(* IEC 61131-3 sources: teller/JD_Teller_LC2_V11/Class/Varan_DataMover (part 2) *)

	//check ASY RD DO's
	for i := 0 to VM_DATAMOVER_MAX_DO - 1 do

		//if handle not exists
		if ( a_DO_ASY_RD[ i ].p_Handle = NIL ) then
			exit;
		end_if;

    ud_retries := VaranIn.GetRetryCounter(ud_DOHandle := a_DO_ASY_RD[ i ].p_Handle$UDINT);
    if ( ud_retries <> a_DO_ASY_RD[ i ].us_OldRetryCounter ) then
      VaranIn.RetryCounter += TO_USINT( ud_retries - a_DO_ASY_RD[ i ].us_OldRetryCounter );
      a_DO_ASY_RD[ i ].us_OldRetryCounter := ud_retries$USINT;
		end_if;
	end_for;

	//check ASY WR DO's
	for i := 0 to VM_DATAMOVER_MAX_DO - 1 do

		//if handle not exists
		if ( a_DO_ASY_WR[ i ].p_Handle = NIL ) then
			exit;
		end_if;

    ud_retries := VaranIn.GetRetryCounter(ud_DOHandle := a_DO_ASY_WR[ i ].p_Handle$UDINT);
    if ( ud_retries <> a_DO_ASY_WR[ i ].us_OldRetryCounter ) then
      VaranIn.RetryCounter += TO_USINT( ud_retries - a_DO_ASY_WR[ i ].us_OldRetryCounter );
      a_DO_ASY_WR[ i ].us_OldRetryCounter := ud_retries$USINT;
		end_if;
	end_for;

	//check config DO
	if ( s_ConfigDO.p_Handle <> NIL ) then

		ud_retries := VaranIn.GetRetryCounter(ud_DOHandle := s_ConfigDO.p_Handle$UDINT);
    if ( ud_retries <> s_ConfigDO.us_OldRetryCounter ) then
      VaranIn.RetryCounter += TO_USINT( ud_retries - s_ConfigDO.us_OldRetryCounter );
      s_ConfigDO.us_OldRetryCounter := ud_retries$USINT;
		end_if;
	end_if;

	//check config DO
	if ( s_ConfigWrDO.p_Handle <> NIL ) then

		//if counter changes
    ud_retries := VaranIn.GetRetryCounter(ud_DOHandle := s_ConfigWrDO.p_Handle$UDINT);
    if ( ud_retries <> s_ConfigWrDO.us_OldRetryCounter ) then
      VaranIn.RetryCounter += TO_USINT( ud_retries - s_ConfigWrDO.us_OldRetryCounter );
      s_ConfigWrDO.us_OldRetryCounter := ud_retries$USINT;
		end_if;
	end_if;

//-------------------------------------------------------------------------------------------------
#ifdef VM_DATAMOVER_ISO_TIME
	//check ISO Time DO
	if ( s_ISO_Time_DO.p_Handle <> NIL ) then

    ud_retries := VaranIn.GetRetryCounter(ud_DOHandle := s_ISO_Time_DO.p_Handle$UDINT);
    if ( ud_retries <> s_ISO_Time_DO.us_OldRetryCounter ) then
      VaranIn.RetryCounter += TO_USINT( ud_retries - s_ISO_Time_DO.us_OldRetryCounter );
      s_ISO_Time_DO.us_OldRetryCounter := ud_retries$USINT;
		end_if;
	end_if;
#endif
//-------------------------------------------------------------------------------------------------

	//----------------we have special DO----------------------------------------------------
	if ( us_specialDOCnt <> 0 ) then

		for i := 0 to us_SpecialDOCnt - 1 do

      ud_retries := VaranIn.GetRetryCounter(ud_DOHandle := a_SpecialDO[ i ].p_Handle$UDINT);
      if ( ud_retries <> a_SpecialDO[ i ].us_OldRetryCounter ) then
        VaranIn.RetryCounter += TO_USINT( ud_retries - a_SpecialDO[ i ].us_OldRetryCounter );
        a_SpecialDO[ i ].us_OldRetryCounter := ud_retries$USINT;
			end_if;
		end_for;
	end_if;

END_FUNCTION //GLOBAL Varan_DataMover::GetRetryCounter
//=================================================================================================
//Function to set off all DO's
//=================================================================================================
FUNCTION GLOBAL Varan_DataMover::SetDOsOff
  VAR
    i		: USINT;
  END_VAR

	//check ISO RD DO's
	for i := 0 to VM_DATAMOVER_MAX_DO - 1 do

		//if handle not exists
		if ( a_DO_ISO_RD[ i ].p_Handle = NIL ) then
			exit;
		end_if;

		//set DO off
    VaranIn.DisableDO(ud_DOHandle := a_DO_ISO_RD[ i ].p_Handle$UDINT);
    a_DO_ISO_RD[ i ].b_DOIsRunning := 0;
	end_for;

	//check ISO WR DO's
	for i := 0 to VM_DATAMOVER_MAX_DO - 1 do

		//if handle not exists
		if ( a_DO_ISO_WR[ i ].p_Handle = NIL ) then
			exit;
		end_if;

		//set DO off
    VaranIn.DisableDO(ud_DOHandle := a_DO_ISO_WR[ i ].p_Handle$UDINT);
    a_DO_ISO_WR[ i ].b_DOIsRunning := 0;
	end_for;

	//check ASY RD DO's
	for i := 0 to VM_DATAMOVER_MAX_DO - 1 do

		//if handle not exists
		if ( a_DO_ASY_RD[ i ].p_Handle = NIL ) then
			exit;
		end_if;

		//set DO off
    VaranIn.DisableDO(ud_DOHandle := a_DO_ASY_RD[ i ].p_Handle$UDINT);
    a_DO_ASY_RD[ i ].b_DOIsRunning := 0;
	end_for;

	//check ASY WR DO's
	for i := 0 to VM_DATAMOVER_MAX_DO - 1 do

		//if handle not exists
		if ( a_DO_ASY_WR[ i ].p_Handle = NIL ) then
			exit;
		end_if;

		//set DO off
    VaranIn.DisableDO(ud_DOHandle := a_DO_ASY_WR[ i ].p_Handle$UDINT);
    a_DO_ASY_WR[ i ].b_DOIsRunning := 0;
	end_for;

	//check config DO
	if ( s_ConfigDO.p_Handle <> NIL ) then

		//set DO off
		VaranIn.DisableDO(ud_DOHandle := s_ConfigDO.p_Handle$UDINT);
	end_if;

	//check config WR DO
	if ( s_ConfigWrDO.p_Handle <> NIL ) then

		//set DO off
		VaranIn.DisableDO(ud_DOHandle := s_ConfigWrDO.p_Handle$UDINT);
    s_ConfigWrDO.b_DOIsRunning := 0;
	end_if;

//-------------------------------------------------------------------------------------------------
#ifdef VM_DATAMOVER_ISO_TIME
	//check ISO Time DO
	if ( s_ISO_Time_DO.p_Handle <> NIL ) then

		//set DO off
		VaranIn.DisableDO(ud_DOHandle := s_ISO_Time_DO.p_Handle$UDINT);
	end_if;
#endif
//-------------------------------------------------------------------------------------------------

	//----------------we have special DO----------------------------------------------------
	if ( us_SpecialDOCnt <> 0 ) then

		for i := 0 to us_SpecialDOCnt - 1 do
			//set DO off
			VaranIn.DisableDO(ud_DOHandle := a_SpecialDO[i].p_Handle$UDINT);
      a_SpecialDO[i].b_DOIsRunning := 0;
		end_for;
	end_if;

END_FUNCTION //GLOBAL Varan_DataMover::SetDOsOff
//=================================================================================================
//Function to start ASY List
//=================================================================================================
FUNCTION  Varan_DataMover::StartAsyncList
  VAR
    i			: USINT;
    StartIt : BOOL;
    lbs_ControlReg : t_MoverConfigReg;
  END_VAR

  // switch off dias alive enable
	s_Config.us_ControlReg.DiasAliveEnable	:= FALSE;

	//if we have ASY DO's
	if ( s_Set_ASY_WR.us_DOCount ) then
		for i := 0 to s_Set_ASY_WR.us_DOCount - 1 do
			//start DO single
      if b_PayloadSupport then
        a_DO_ASY_WR[ i ].b_DOIsRunning.StartRequest := TRUE;
      else
      a_DO_ASY_WR[ i ].p_Handle^.ucCtrlStat := VaranIn.SetRunStatus(VARAN_DO_SINGLE_RUN);
      end_if;
		end_for;
	end_if;

  StartIt := FALSE;
	//if we have ASY code
	if ( ui_ASYByteCount ) then
  	//start async list
    s_Config.us_ControlReg.AsyncListEnable	:= TRUE;
    StartIt := TRUE;
  else
  	//don't start async list
    s_Config.us_ControlReg.AsyncListEnable	:= FALSE;

    // if there is no ASY code => don't wait for anything
    us_Wait := 0;
  end_if;
  lbs_ControlReg := s_Config.us_ControlReg;

  if ( lbs_ControlReg.AdminEnable = TRUE ) then
    b_AdminStarted := TRUE;
    us_ControlRd.AdminActive := TRUE;
    StartIt := TRUE;
  end_if;

  if StartIt then
    s_ConfigWrDO.p_DataWrite^ := lbs_ControlReg;

    // reset flag for starting admin task
    IF lbs_ControlReg.AdminEnable = TRUE THEN
      s_Config.us_ControlReg.AdminEnable := FALSE;
    END_IF;

    if b_PayloadSupport then
      s_ConfigWrDO.b_DOIsRunning.StartRequest :=TRUE;
    else
    s_ConfigWrDO.p_Handle^.ucCtrlStat := VaranIn.SetRunStatus(VARAN_DO_SINGLE_RUN);
    end_if;
		us_Wait := 1;		//because otherwise we have old async ready bit

	end_if;

END_FUNCTION // Varan_DataMover::StartAsyncList
//[#ENGLISH]
//=================================================================================================
//Function to add an ISO Rd Enable
//=================================================================================================
//[>ud_add]address of access
//[>ud_length]length of data
//[>p_data]address of pointer variable to save data address
//[>p_enable]address of pointer to start single call
FUNCTION GLOBAL Varan_DataMover::AddRdISOEnable
  VAR_INPUT
    ud_add			: UDINT;
    ud_length		: UDINT;
    p_data			: ^void;
    p_enable		: ^USINT;
      ud_Priority 	: HDINT;
    p_DataAddr : ^HDINT;
		p_UserDOHandle 	: ^UDINT;
  END_VAR
  VAR_OUTPUT
    sd_retval		: DINT;
  END_VAR
  VAR
    p_Mov			: ^t_StructMoveEn;
    ud_dest_add		: UDINT;
    ud_en_add		: UDINT;
  END_VAR

	//get memory for single call
  sd_retval := GetMemoryISORd(p_add         := #ud_dest_add
                              , p_data	:= p_data
                              , ud_len	:= ud_length
                              , ud_Priority := ud_Priority
                            , p_UserDOHandle:= p_UserDOHandle
                              );

	if ( sd_retval <> VARANMANAGER_OK ) then
		return;
	end_if;

  //give back the address if requested
  if p_DataAddr then
    p_DataAddr^ := ud_dest_add;
  end_if;

	//for enable byte
	sd_retval := GetMemoryISOWr	( p_add		:= #ud_en_add
                              , p_data	:= p_enable
                              , ud_len	:= 1
                              );

	if ( sd_retval <> VARANMANAGER_OK ) then
		return;
	end_if;

	//give back address of enable byte
	( ( ( p_enable$^UDINT )^ )$^USINT )^ := 0;

	//save opcodes in class
	if ( p_ISOMoverCode = NIL ) then
		//allocate memory
		p_ISOMoverCode$^void := To_StdLib.Malloc( s_Set_ISO_RD.ui_DPRAMSize + s_Set_ISO_WR.ui_DPRAMSize );

		if ( p_ISOMoverCode  = NIL ) then
			State := _MemoryFault;
			sd_retval := -103;
			VaranIn.SetState( State );
			return;
		end_if;
	end_if;

	//first check length
	if ( CheckLengthOfCode() = FALSE ) then
		sd_retval := -102;
		return;
	end_if;

	//check size of free memory
	if (( ui_ISOByteCount + sizeof( t_StructMoveEn )) > ( s_Set_ISO_RD.ui_DPRAMSize + s_Set_ISO_WR.ui_DPRAMSize )) then
		State := _MemoryFault;
		sd_retval := -102;
		VaranIn.SetState( State );
		return;
	end_if;

	//get right pointer
	p_Mov := p_ISOMoverCode + ui_ISOByteCount;

	p_Mov^.us_Command 		:= VM_DATAMOVER_MOVE_EN_OP;
	p_Mov^.ui_Length		:= ud_length$UINT;
	p_Mov^.us_Length		:= ( ud_length shr 16 )$USINT;
	p_Mov^.ud_SourceAdd		:= ud_add;
	p_Mov^.ud_DestAdd		:= ud_dest_add;
	p_Mov^.ud_EnableAddByte	:= ud_en_add;

	ui_ISOByteCount += sizeof( t_StructMoveEn );

	sd_retval := VARANMANAGER_OK;

END_FUNCTION //GLOBAL Varan_DataMover::AddRdISOSingle
//[#ENGLISH]
//=================================================================================================
//Function to add an ISO Wr Enable
//=================================================================================================
//[>ud_add]address of access
//[>ud_length]length of data
//[>p_data]address of pointer variable to save data address
//[>p_enable]address of pointer to start single call
FUNCTION GLOBAL Varan_DataMover::AddWrISOEnable
  VAR_INPUT
    ud_add			: UDINT;
    ud_length		: UDINT;
    p_data			: ^void;
    p_enable		: ^USINT;
      ud_Priority 	: HDINT;
    p_DataAddr : ^HDINT;
		p_UserDOHandle 	: ^UDINT;
  END_VAR
  VAR_OUTPUT
    sd_retval		: DINT;
  END_VAR
  VAR
    p_Mov			: ^t_StructMoveEn;
    ud_dest_add		: UDINT;
  END_VAR

	//get memory for write single call (+1 because of enable byte)
  sd_retval := GetMemoryISOWr(p_add         := #ud_dest_add
                              , p_data	:= p_data
                              , ud_len	:= ud_length + 1
                              , ud_Priority := ud_Priority
                            , p_UserDOHandle:= p_UserDOHandle
                              );

	if ( sd_retval <> VARANMANAGER_OK ) then
		return;
	end_if;

  //give back the address if requested
  if p_DataAddr then
    p_DataAddr^ := ud_dest_add;
  end_if;

	//give back address of enable byte
	( p_enable$^UDINT )^ := ( p_data$^UDINT )^ + ud_length;
	( ( ( p_enable$^UDINT )^ )$^USINT )^ := 0;

	//save opcodes in class
	if ( p_ISOMoverCode = NIL ) then
		//allocate memory
		p_ISOMoverCode$^void := To_StdLib.Malloc( s_Set_ISO_WR.ui_DPRAMSize + s_Set_ISO_RD.ui_DPRAMSize );

		if ( p_ISOMoverCode = NIL ) then
			State := _MemoryFault;
			sd_retval := -103;
			VaranIn.SetState( State );
			return;
		end_if;
	end_if;

	//first check length
	if ( CheckLengthOfCode() = FALSE ) then
		sd_retval := -102;
		return;
	end_if;

	//check size of free memory
	if (( ui_ISOByteCount + sizeof( t_StructMoveEn )) > ( s_Set_ISO_RD.ui_DPRAMSize + s_Set_ISO_WR.ui_DPRAMSize )) then
		State := _MemoryFault;
		sd_retval := -102;
		VaranIn.SetState( State );
		return;
	end_if;

	//get right pointer
	p_Mov := p_ISOMoverCode + ui_ISOByteCount;

	p_Mov^.us_Command 		:= VM_DATAMOVER_MOVE_EN_OP;
	p_Mov^.ui_Length		:= ud_length$UINT;
	p_Mov^.us_Length		:= ( ud_length shr 16 )$USINT;
	p_Mov^.ud_SourceAdd		:= ud_dest_add;
	p_Mov^.ud_DestAdd		:= ud_add;
	p_Mov^.ud_EnableAddByte	:= ud_dest_add + ud_length;

	ui_ISOByteCount += sizeof( t_StructMoveEn );

	sd_retval := VARANMANAGER_OK;

END_FUNCTION //GLOBAL Varan_DataMover::AddWrISOSingle
//[#ENGLISH]
//=================================================================================================
//Function to add an ASY Rd Enable
//=================================================================================================
//[>ud_add]address of access
//[>ud_length]length of data
//[>p_data]address of pointer variable to save data address
//[>p_enable]address of pointer to start single call
FUNCTION GLOBAL Varan_DataMover::AddRdASYEnable
  VAR_INPUT
    ud_add			: UDINT;
    ud_length		: UDINT;
    p_data			: ^void;
    p_enable		: ^USINT;
      ud_Priority 	: HDINT;
    p_DataAddr : ^HDINT;
		p_UserDOHandle 	: ^UDINT;
  END_VAR
  VAR_OUTPUT
    sd_retval		: DINT;
  END_VAR
  VAR
    p_Mov			: ^t_StructMoveEn;
    ud_dest_add		: UDINT;
    ud_en_add		: UDINT;
  END_VAR

	//get memory for write single call
  sd_retval := GetMemoryASYRd(p_add         := #ud_dest_add
                              , p_data	:= p_data
                              , ud_len	:= ud_length
                              , ud_Priority := ud_Priority
                            , p_UserDOHandle:=p_UserDOHandle
                              );

	if ( sd_retval <> VARANMANAGER_OK ) then
		return;
	end_if;

  //give back the address if requested
  if p_DataAddr then
    p_DataAddr^ := ud_dest_add;
  end_if;

	//for enable byte
	sd_retval := GetMemoryASYWr	( p_add		:= #ud_en_add
                              , p_data	:= p_enable
                              , ud_len	:= 1
                              , ud_Priority := ud_Priority
                              );

	if ( sd_retval <> VARANMANAGER_OK ) then
		return;
	end_if;

	//give back address of enable byte
	( ( ( p_enable$^UDINT )^ )$^USINT )^ := 0;

	//save opcodes in class
	if ( p_ASYMoverCode = NIL ) then
		//allocate memory
		p_ASYMoverCode$^void := To_StdLib.Malloc( s_Set_ASY_RD.ui_DPRAMSize + s_Set_ASY_WR.ui_DPRAMSize );

		if ( p_ASYMoverCode  = NIL ) then
			State := _MemoryFault;
			sd_retval := -103;
			VaranIn.SetState( State );
			return;
		end_if;
	end_if;

	//first check length
	if ( CheckLengthOfCode() = FALSE ) then
		sd_retval := -102;
		return;
	end_if;

	//check size of free memory
	if (( ui_ASYByteCount + sizeof( t_StructMoveEn )) > ( s_Set_ASY_RD.ui_DPRAMSize + s_Set_ASY_WR.ui_DPRAMSize )) then
		State := _MemoryFault;
		sd_retval := -102;
		VaranIn.SetState( State );
		return;
	end_if;

	//get right pointer
	p_Mov := p_ASYMoverCode + ui_ASYByteCount;

	p_Mov^.us_Command 		:= VM_DATAMOVER_MOVE_EN_OP;
	p_Mov^.ui_Length		:= ud_length$UINT;
	p_Mov^.us_Length		:= ( ud_length shr 16 )$USINT;
	p_Mov^.ud_SourceAdd		:= ud_add;
	p_Mov^.ud_DestAdd		:= ud_dest_add;
	p_Mov^.ud_EnableAddByte	:= ud_en_add;

	ui_ASYByteCount += sizeof( t_StructMoveEn );

	sd_retval := VARANMANAGER_OK;

END_FUNCTION //GLOBAL Varan_DataMover::AddRdASYEnable
//[#ENGLISH]
//=================================================================================================
//Function to add an ASY Wr Enable
//=================================================================================================
//[>ud_add]address of access
//[>ud_length]length of data
//[>p_data]address of pointer variable to save data address
//[>p_enable]address of pointer to start single call
FUNCTION GLOBAL Varan_DataMover::AddWrASYEnable
  VAR_INPUT
    ud_add			: UDINT;
    ud_length		: UDINT;
    p_data			: ^void;
    p_enable		: ^USINT;
    ud_Priority 	: HDINT;
    p_DataAddr : ^HDINT;
		p_UserDOHandle 	: ^UDINT;
  END_VAR
  VAR_OUTPUT
    sd_retval		: DINT;
  END_VAR
  VAR
    p_Mov			: ^t_StructMoveEn;
    ud_dest_add		: UDINT;
  END_VAR

	//get memory for write single call (+1 because of enable byte)
  sd_retval := GetMemoryASYWr(p_add         := #ud_dest_add
                              , p_data	:= p_data
                              , ud_len	:= ud_length + 1
                              , ud_Priority := ud_Priority
                            , p_UserDOHandle:= p_UserDOHandle
                              );

	if ( sd_retval <> VARANMANAGER_OK ) then
		return;
	end_if;

  //give back the address if requested
  if p_DataAddr then
    p_DataAddr^ := ud_dest_add;
  end_if;

	//give back address of enable byte
	( p_enable$^UDINT )^ := ( p_data$^UDINT )^ + ud_length;
	( ( ( p_enable$^UDINT )^ )$^USINT )^ := 0;

	//save opcodes in class
	if ( p_ASYMoverCode = NIL ) then
		//allocate memory
		p_ASYMoverCode$^void := To_StdLib.Malloc( s_Set_ASY_WR.ui_DPRAMSize + s_Set_ASY_RD.ui_DPRAMSize );

		if ( p_ASYMoverCode = NIL ) then
			State := _MemoryFault;
			sd_retval := -103;
			VaranIn.SetState( State );
			return;
		end_if;
	end_if;

	//first check length
	if ( CheckLengthOfCode() = FALSE ) then
		sd_retval := -102;
		return;
	end_if;

	//check size of free memory
	if (( ui_ASYByteCount + sizeof( t_StructMoveEn )) > ( s_Set_ASY_RD.ui_DPRAMSize + s_Set_ASY_WR.ui_DPRAMSize )) then
		State := _MemoryFault;
		sd_retval := -102;
		VaranIn.SetState( State );
		return;
	end_if;

	//get right pointer
	p_Mov := p_ASYMoverCode + ui_ASYByteCount;

	p_Mov^.us_Command 		:= VM_DATAMOVER_MOVE_EN_OP;
	p_Mov^.ui_Length		:= ud_length$UINT;
	p_Mov^.us_Length		:= ( ud_length shr 16 )$USINT;
	p_Mov^.ud_SourceAdd		:= ud_dest_add;
	p_Mov^.ud_DestAdd		:= ud_add;
	p_Mov^.ud_EnableAddByte	:= ud_dest_add + ud_length;

	ui_ASYByteCount += sizeof( t_StructMoveEn );

	sd_retval := VARANMANAGER_OK;

END_FUNCTION //GLOBAL Varan_DataMover::AddWrASYSingle
//[#ENGLISH]
//=================================================================================================
//Function to get next free space for ISO read
//=================================================================================================
//[>p_add]value for destination address
//[>p_data]pointer to data in DO
//[>ud_len]length of data
FUNCTION  Varan_DataMover::GetMemoryISORd
  VAR_INPUT
    p_add			: ^UDINT;
    p_data			: ^void;
    ud_len			: UDINT;
    ud_Priority 	: HDINT;
    p_UserDOHandle 	: ^UDINT;
  END_VAR
  VAR_OUTPUT
    sd_retval		: DINT;
  END_VAR
  VAR
    p_DO			: ^t_DO_RD;
    i				: UINT;
  END_VAR

	sd_retval := 0;
	p_DO := NIL;

	//not more than 128 Byte
	if ( ud_len > 128 ) then
		sd_retval := -100;
		return;
	end_if;

	//search for free space
	if ( s_Set_ISO_RD.us_DOCount ) then
		for i := 0 to s_Set_ISO_RD.us_DOCount - 1 do
			if ( a_DO_ISO_RD[ i ].us_Length + ud_len <= 128 ) then
				p_DO := #a_DO_ISO_RD[ i ];
				p_add^ := ( i * 128 ) + p_DO^.us_Length + s_Set_ISO_RD.ui_DPRAMOffsetSub;
				exit;
			end_if;
		end_for;
	end_if;

	//if no space create DO
	if ( p_DO = NIL ) then

    //#WP003 start
    //check for error -> after creation, no DO change is possible
    if DO_Created then
      State := _CreateDOFailed;
      VaranIn.SetState( State );
      return;
    end_if;

    //check if we have enough space
    if ( s_Set_ISO_RD.ui_DPRAMSize / 128 <= s_Set_ISO_RD.us_DOCount ) then
      sd_retval := -101;
      State := _MemoryFault;
      VaranIn.SetState( State );
      return;
    end_if;

    p_DO := #a_DO_ISO_RD[ s_Set_ISO_RD.us_DOCount ];
	  p_add^ := s_Set_ISO_RD.us_DOCount * 128 + s_Set_ISO_RD.ui_DPRAMOffsetSub;
	  s_Set_ISO_RD.us_DOCount += 1;
	end_if;

	//give back data pointer of DO
	( p_data$^UDINT )^ := p_DO^.p_DataRead$UDINT + p_DO^.us_Length;

	//set new length of DO
	p_DO^.us_Length += ud_len$USINT;

  // save the priority with the DO
  p_DO^.ud_Priority := ud_Priority;

  // save pointer to save the DO Handle to
  p_DO^.p_UserDOHandle := p_UserDOHandle;

  //WP003 start
  //if first callback give back data-pointer to dummy memory area
  if DO_Created = 0 then
    p_DO^.p_DataRead := p_DummyDataRdWr;
    ( p_data$^UDINT )^ := p_DO^.p_DataRead$UDINT;
  end_if;
  //WP003 end
END_FUNCTION // Varan_DataMover::GetMemoryISORd
//[#ENGLISH]
//=================================================================================================
//Function to get next free space for ISO write
//=================================================================================================
//[>p_add]value for destination address
//[>p_data]pointer to data in DO
//[>ud_len]length of data
FUNCTION  Varan_DataMover::GetMemoryISOWr
  VAR_INPUT
    p_add		: ^UDINT;
    p_data		: ^void;
    ud_len		: UDINT;
    ud_Priority 	: HDINT;
    p_UserDOHandle 	: ^UDINT;
  END_VAR
  VAR_OUTPUT
    sd_retval		: DINT;
  END_VAR
  VAR
    p_DO			: ^t_DO_WR;
    i				: UINT;
  END_VAR

	sd_retval := 0;
	p_DO := NIL;

	//not more than 128 Byte
	if ( ud_len > 128 ) then
		sd_retval := -100;
		return;
	end_if;

	//search for free space
	if ( s_Set_ISO_WR.us_DOCount ) then
		for i := 0 to s_Set_ISO_WR.us_DOCount - 1 do
			if ( a_DO_ISO_WR[ i ].us_Length + ud_len <= 128 ) then
				p_DO := #a_DO_ISO_WR[ i ];
				p_add^ := ( i * 128 ) + p_DO^.us_Length + s_Set_ISO_WR.ui_DPRAMOffsetSub;
				exit;
			end_if;
		end_for;
	end_if;

	//if no space create new DO
	if ( p_DO = NIL ) then

    //#WP003 start
    //check for error -> after creation, no DO change is possible
    if DO_Created then
      State := _CreateDOFailed;
      VaranIn.SetState( State );
      return;
    end_if;

		//check if we have enough space
		if ( s_Set_ISO_WR.ui_DPRAMSize / 128 <= s_Set_ISO_WR.us_DOCount ) then
			sd_retval := -101;
			State := _MemoryFault;
			VaranIn.SetState( State );
			return;
		end_if;
    //#WP003 end

		p_DO := #a_DO_ISO_WR[ s_Set_ISO_WR.us_DOCount ];
		p_add^ := s_Set_ISO_WR.us_DOCount * 128 + s_Set_ISO_WR.ui_DPRAMOffsetSub;
		s_Set_ISO_WR.us_DOCount += 1;
	end_if;

	//give back data pointer of DO
	( p_data$^UDINT )^ := p_DO^.p_DataWrite$UDINT + p_DO^.us_Length;

	//set new length of DO
	p_DO^.us_Length += ud_len$USINT;

  // save the priority with the DO
  p_DO^.ud_Priority := ud_Priority;

  // save pointer to save the DO Handle to
  p_DO^.p_UserDOHandle := p_UserDOHandle;

  //WP003 start
  //if first callback give back data-pointer to dummy memory area
  if DO_Created = 0 then
    p_DO^.p_DataWrite := p_DummyDataRdWr;
    ( p_data$^UDINT )^ := p_DO^.p_DataWrite$UDINT;
  end_if;
  //WP003 end
END_FUNCTION // Varan_DataMover::GetMemoryISOWr
//[#ENGLISH]
//=================================================================================================
//Function to get next free space for ASY read
//=================================================================================================
//[>p_add]value for destination address
//[>p_data]pointer to data in DO
//[>ud_len]length of data
FUNCTION  Varan_DataMover::GetMemoryASYRd
  VAR_INPUT
    p_add		: ^UDINT;
    p_data		: ^void;
    ud_len		: UDINT;
    ud_Priority 	: HDINT;
    p_UserDOHandle 	: ^UDINT;
  END_VAR
  VAR_OUTPUT
    sd_retval		: DINT;
  END_VAR
  VAR
    p_DO			: ^t_DO_RD;
    i				: UINT;
  END_VAR

	sd_retval := 0;
	p_DO := NIL;

	//not more than 128 Byte
	if ( ud_len > 128 ) then
		sd_retval := -100;
		return;
	end_if;

	p_DO := NIL;

	//search for free space
	if ( s_Set_ASY_RD.us_DOCount ) then
		for i := 0 to s_Set_ASY_RD.us_DOCount - 1 do
			if ( a_DO_ASY_RD[ i ].us_Length + ud_len <= 128 ) then
				p_DO := #a_DO_ASY_RD[ i ];
				p_add^ := ( i * 128 ) + p_DO^.us_Length + s_Set_ASY_RD.ui_DPRAMOffsetSub;
				exit;
			end_if;
		end_for;
	end_if;

	//if no space in DOs allocate new DO
	if ( p_DO = NIL ) then

      //#WP003 start
      //check for error -> after creation, no DO change is possible
      if DO_Created then
        State := _CreateDOFailed;
	    VaranIn.SetState( State );
	    return;
      end_if;

	  //check if we have enough space
	  if ( s_Set_ASY_RD.ui_DPRAMSize / 128 <= s_Set_ASY_RD.us_DOCount ) then
		sd_retval := -101;
		State := _MemoryFault;
		VaranIn.SetState( State );
		return;
	  end_if;
      //#WP003 end

	  p_DO := #a_DO_ASY_RD[ s_Set_ASY_RD.us_DOCount ];
	  p_add^ := s_Set_ASY_RD.us_DOCount * 128 + s_Set_ASY_RD.ui_DPRAMOffsetSub;
	  s_Set_ASY_RD.us_DOCount += 1;
    end_if;

	//give back data pointer of DO
	( p_data$^UDINT )^ := p_DO^.p_DataRead$UDINT + p_DO^.us_Length;

	//set new length of DO
	p_DO^.us_Length += ud_len$USINT;

  // save the priority with the DO
  p_DO^.ud_Priority := ud_Priority;

  // save pointer to save the DO Handle to
  p_DO^.p_UserDOHandle := p_UserDOHandle;

  //WP003 start
  //if first callback give back data-pointer to dummy memory area
  if DO_Created = 0 then
    p_DO^.p_DataRead := p_DummyDataRdWr;
    ( p_data$^UDINT )^ := p_DO^.p_DataRead$UDINT;
  end_if;
  //WP003 end

END_FUNCTION // Varan_DataMover::GetMemoryASYRd
//[#ENGLISH]
//=================================================================================================
//Function to get next free space for ASY write
//=================================================================================================
//[>p_add]value for destination address
//[>p_data]pointer to data in DO
//[>ud_len]length of data
FUNCTION  Varan_DataMover::GetMemoryASYWr
  VAR_INPUT
    p_add		: ^UDINT;
    p_data		: ^void;
    ud_len		: UDINT;
      ud_Priority 	: HDINT;
    p_UserDOHandle 	: ^UDINT;
  END_VAR
  VAR_OUTPUT
    sd_retval		: DINT;
  END_VAR
  VAR
    p_DO			: ^t_DO_WR;
    i				: UINT;
  END_VAR

	sd_retval := 0;
	p_DO := NIL;

	//not more than 128 Byte
	if ( ud_len > 128 ) then
		sd_retval := -100;
		return;
	end_if;

	//search for free space
	if ( s_Set_ASY_WR.us_DOCount ) then
		for i := 0 to s_Set_ASY_WR.us_DOCount - 1 do
			if ( a_DO_ASY_WR[ i ].us_Length + ud_len <= 128 ) then
				p_DO := #a_DO_ASY_WR[ i ];
				p_add^ := ( i * 128 ) + p_DO^.us_Length + s_Set_ASY_WR.ui_DPRAMOffsetSub;
				exit;
			end_if;
		end_for;
	end_if;

  //if no space in DOs allocate new DO
  if ( p_DO = NIL ) then

  //#WP003 start
  //check for error -> after creation, no DO change is possible
    if DO_Created then
      State := _CreateDOFailed;
      VaranIn.SetState( State );
      return;
    end_if;

	  //check if we have enough space
	  if ( s_Set_ASY_WR.ui_DPRAMSize / 128 <= s_Set_ASY_WR.us_DOCount ) then
      sd_retval := -101;
      State := _MemoryFault;
      VaranIn.SetState( State );
      return;
	  end_if;
      //#WP003 end

	  p_DO := #a_DO_ASY_WR[ s_Set_ASY_WR.us_DOCount ];
	  p_add^ := s_Set_ASY_WR.us_DOCount * 128 + s_Set_ASY_WR.ui_DPRAMOffsetSub;
	  s_Set_ASY_WR.us_DOCount += 1;
	end_if;

	//give back data pointer of DO
	( p_data$^UDINT )^ := p_DO^.p_DataWrite$UDINT + p_DO^.us_Length;

	//set new length of DO
	p_DO^.us_Length += ud_len$USINT;

  // save the priority with the DO
  p_DO^.ud_Priority := ud_Priority;

  // save pointer to save the DO Handle to
  p_DO^.p_UserDOHandle := p_UserDOHandle;

  //WP003 start
  //if first callback give back data-pointer to dummy memory area
  if DO_Created = 0 then
    p_DO^.p_DataWrite := p_DummyDataRdWr;
    ( p_data$^UDINT )^ := p_DO^.p_DataWrite$UDINT;
  end_if;
  //WP003 end

END_FUNCTION // Varan_DataMover::GetMemoryASYWr
//[#ENGLISH]
//=================================================================================================
//Function to set DIAS Alvie Signal Address
//=================================================================================================
//[>ud_address]address of dias module
FUNCTION GLOBAL Varan_DataMover::SetDiasAliveSignal
  VAR_INPUT
    ud_address		: UDINT;
    us_mode			: USINT;
  END_VAR
  VAR_OUTPUT
    sd_retval		: DINT;
  END_VAR
  VAR
    a_data			: ARRAY[0..4] OF USINT;
  END_VAR

	a_data[ 0 ]$UDINT := ud_address;
	a_data[ 4 ] := us_mode;
  if b_PayloadSupport then
    //write config data (because we need direct accesses in init)
    sd_retval := MULTI_VARAN_iExecuteDirectAccess(hNodeHandle := ud_HandleModule
                                                , udCommand   := VARAN_CMD_MEMORY_WRITE
                                                , udOffset    := CodeStartAddress + VM_DATAMOVER_DIAS_ALIVE
                                                , udLength    := sizeof(  a_data )
                                                , pusData     := ( #a_data )$^USINT
                                                , pudErrorInfo:= NIL);

    if ( sd_retval <> VARANMANAGER_OK ) then
      State := _DirectAccessFailed;
      VaranIn.SetState( State );
      return;
    end_if;

    s_Config.us_ControlReg.DiasAliveEnable := TRUE;

    //write config data (because we need direct accesses in init)
    sd_retval := MULTI_VARAN_iExecuteDirectAccess(hNodeHandle := ud_HandleModule
                                                , udCommand   := VARAN_CMD_MEMORY_WRITE
                                                , udOffset    := CodeStartAddress
                                                , udLength    := sizeof( t_DataMoverConfig )
                                                , pusData     := ( #s_Config )$^USINT
                                                , pudErrorInfo:= NIL);

    if ( sd_retval <> VARANMANAGER_OK ) then
      State := _DirectAccessFailed;
      VaranIn.SetState( State );
      return;
    end_if;

  else
    //write config data (because we need direct accesses in init)
    sd_retval := VARAN_iWriteMemoryDA(uiManager     := ud_VaranManagerNr
                                    , uiAddress     := ud_DeviceAddress + CodeStartAddress + VM_DATAMOVER_DIAS_ALIVE
                                    , uiLen         := sizeof( a_data )
                                    , uiRetryTimeout:= s_DAData.ud_RetryTimeout
                                    , pvData        := #a_data
                                    , puiError      := NIL
                                    );

    if ( sd_retval <> VARANMANAGER_OK ) then
      State := _DirectAccessFailed;
      VaranIn.SetState( State );
      return;
    end_if;

    s_Config.us_ControlReg.DiasAliveEnable := TRUE;

    //write config data (because we need direct accesses in init)
    sd_retval := VARAN_iWriteMemoryDA(uiManager     := ud_VaranManagerNr
                                    , uiAddress     := ud_DeviceAddress + CodeStartAddress
                                    , uiLen         := sizeof( t_DataMoverConfig )
                                    , uiRetryTimeout:= VaranIn.GetRetryTimeout( ud_bytes := sizeof( t_DataMoverConfig ) )
                                    , pvData        := #s_Config
                                    , puiError      := NIL
                                     );

    if ( sd_retval <> VARANMANAGER_OK ) then
      State := _DirectAccessFailed;
      VaranIn.SetState( State );
      return;
    end_if;
  end_if;

END_FUNCTION //GLOBAL Varan_DataMover::SetDiasAliveSignal
//=================================================================================================
//Function check if we have enough code space
//=================================================================================================
FUNCTION  Varan_DataMover::CheckLengthOfCode
  VAR_OUTPUT
    b_available		: BOOL;
  END_VAR

	b_available := TRUE;

	//check length
	if ( ui_ISOByteCount + ui_ASYByteCount + sizeof( t_StructMove ) + sizeof( t_StructEnd ) > ( CodeSize - VM_DATAMOVER_CODE_OFFEST ) ) then
		State := _MemoryFault;
		VaranIn.SetState( State );
		b_available := FALSE;
		return;
	end_if;

END_FUNCTION // Varan_DataMover::CheckLengthOfCode
//[#ENGLISH]
//=================================================================================================
//Function to write code to DPRAM
//=================================================================================================
//[>ud_address]address where code should be written
//[>ud_length]length of code
//[>p_data]pointer to data
FUNCTION  Varan_DataMover::WriteCode
  VAR_INPUT
    ud_address		: UDINT;
    ud_length		: UDINT;
    p_data			: ^UDINT;
  END_VAR
  VAR_OUTPUT
    sd_retval		: DINT;
  END_VAR
  VAR
    ud_cnt			: UDINT;
  END_VAR

	//first set fault
	sd_retval := -100;
	ud_cnt := 0;

	//while bytes are available
	while ( ud_length ) do

		//if we have more than 128 bytes or exactly 128 bytes
		if ( ud_length >= 128 ) then
      if b_PayloadSupport then
			//write with direct access
        sd_retval := MULTI_VARAN_iExecuteDirectAccess(hNodeHandle := ud_HandleModule
                                                , udCommand   := VARAN_CMD_MEMORY_WRITE
                                                    , udOffset    := (ud_address + ( ud_cnt * 128 )) and 16#FFFF // Remove DeviceAddress so that offset remains
                                                    , udLength    := 128
                                                    , pusData     := ( p_data + ( ud_cnt * 128 ))$^USINT
                                                , pudErrorInfo:= NIL);

        //look for error
        if ( sd_retval <> VARANMANAGER_OK ) then
          State := _DirectAccessFailed;
          VaranIn.SetState( State );
          return;
        end_if;
      else
        sd_retval := VARAN_iWriteMemoryDA	( uiManager     := ud_VaranManagerNr
                                          , uiAddress     := ud_address + ( ud_cnt * 128 )
                                          , uiLen         := 128
                                        , uiRetryTimeout:= VaranIn.GetRetryTimeout( ud_bytes := 128 ) //s_DAData.ud_RetryTimeout
                                          , pvData        := p_data + ( ud_cnt * 128 )
                                          , puiError      := NIL
                                        );

			//look for error
			if ( sd_retval <> VARANMANAGER_OK ) then
				State := _DirectAccessFailed;
				VaranIn.SetState( State );
				return;
			end_if;
      end_if;

			ud_length -= 128;
			ud_cnt += 1;

		else
      if b_PayloadSupport then
        //write with direct access
        sd_retval := MULTI_VARAN_iExecuteDirectAccess(hNodeHandle := ud_HandleModule
                                                , udCommand   := VARAN_CMD_MEMORY_WRITE
                                                    , udOffset    := (ud_address + ( ud_cnt * 128 )) and 16#FFFF // Remove DeviceAddress so that offset remains
                                                , udLength    := ud_length
                                                    , pusData     := ( p_data + ( ud_cnt * 128 ))$^USINT
                                                , pudErrorInfo:= NIL);

        //look for error
        if ( sd_retval <> VARANMANAGER_OK ) then
          State := _DirectAccessFailed;
          VaranIn.SetState( State );
          return;
        end_if;
      else

			//write rest with direct access
        sd_retval := VARAN_iWriteMemoryDA(uiManager     := ud_VaranManagerNr
                                        , uiAddress     := ( ud_address + ( ud_cnt * 128 ))
                                        , uiLen         := ( ud_length )
                                        , uiRetryTimeout:= VaranIn.GetRetryTimeout( ud_bytes := ud_length ) //s_DAData.ud_RetryTimeout - doesn`t work with CIV 513 => -27
                                        , pvData        := p_data + ( ud_cnt * 128 )
                                        , puiError      := NIL
                                        );

			//look for error
			if ( sd_retval <> VARANMANAGER_OK ) then
				State := _DirectAccessFailed;
				VaranIn.SetState( State );
				return;
			end_if;
		  end_if;
			ud_length := 0;
		end_if;
	end_while;

	//everything OK
	sd_retval := 0;

END_FUNCTION // Varan_DataMover::WriteCode
//[#ENGLISH]
//=================================================================================================
//Function to get actual pointer to code address
//=================================================================================================
//[>ud_type] Bit31: get pointer to ISO code in heap, Bit30: get code start address (available after connect), else actual ISO Byte count
FUNCTION GLOBAL Varan_DataMover::GetActualAddressPointerISO
  VAR_INPUT
    ud_type		: UDINT;
  END_VAR
  VAR_OUTPUT
    ud_add_off		: UDINT;
  END_VAR

	//if type is set we return mover code pointer in heap
	if ( ud_type and 16#8000_0000 ) then
		ud_add_off := p_ISOMoverCode$UDINT;

	//or get code start address (valid after Connect function)
	elsif ( ud_type and 16#4000_0000 ) then
		ud_add_off := CodeStartAddress + s_ListSettings.ui_SyncListStart;

	//otherwise we return actual offset in Code DPRAM
	else
		ud_add_off := ui_ISOByteCount;
	end_if;

END_FUNCTION //GLOBAL Varan_DataMover::GetActualAddressPointerISO
//[#ENGLISH]
//=================================================================================================
//Function to get actual pointer to code address
//=================================================================================================
FUNCTION GLOBAL Varan_DataMover::GetActualAddressPointerASY
  VAR_INPUT
    ud_type		: UDINT;
  END_VAR
  VAR_OUTPUT
    ud_add_off		: UDINT;
  END_VAR

	//if type is set we return mover code pointer in heap
	if ( ud_type and 16#8000_0000 ) then
		ud_add_off := p_ASYMoverCode$UDINT;

	//or get code start address (valid after Connect function)
	elsif ( ud_type and 16#4000_0000 ) then
		ud_add_off := CodeStartAddress + s_ListSettings.ui_AsyncListStart;

	//otherwise we return actual offset in Code DPRAM
	else
		ud_add_off := ui_ASYByteCount;
	end_if;

END_FUNCTION //GLOBAL Varan_DataMover::GetActualAddressPointerASY
//[#ENGLISH]
//=================================================================================================
//Function to install special write DO (for CRIF)
//=================================================================================================
//[>ud_dol_type] pointer to variable to set right handle
//[>p_ud_handle]pointer to variable to set right handle
//[>ud_address] Address of data object
//[>ud_length] Length of data object
//[>p_ud_data] pointer to variable to get pointer to data
//[>ud_type]0=control area, 1=memory area
//[<sd_retval] 0=OK, negative=error (look lsl_st_varan.h)
FUNCTION GLOBAL Varan_DataMover::AddVaranWrDO
  VAR_INPUT
    ud_dol_type		: UDINT;
    p_ud_handle		: ^UDINT;
    ud_address		: UDINT;
    ud_length		: UDINT;
    p_ud_data		: ^UDINT;
    ud_type			: UDINT;
  END_VAR
  VAR_OUTPUT
    sd_retval		: DINT;
  END_VAR

	//check number
	if ( us_SpecialDOCnt > 10 ) then
		sd_retval := -100;
		return;
	end_if;

	//create special DO
  if b_PayloadSupport then

    sd_retval := VaranIn.AddWrPayloadDO(ud_dol_type     := ud_dol_type
                                      , p_ud_handle     := p_ud_handle
                                      , ud_offset_write := ud_address and 16#FFFF // Mask out die DeviceAddress
                                      , ud_length_write := ud_length
                                      , p_ud_data_write := p_ud_data
                                      , ud_type         := VM_MEMORY_ACCESS
                                      );

    //look if an error occurs
    if ( sd_retval <> VARANMANAGER_OK ) then
      State := _CreateDOFailed;
      VaranIn.SetState( State );
      return;
    end_if;

  else
    sd_retval := VaranIn.VaranIn.AddWrDO( p_us_position_info:= p_NodeString
                                      , ud_dol_type			:= ud_dol_type
                                      , p_ud_handle			:= p_ud_handle
                                      , ud_address			:= ud_address
                                      , ud_length				:= ud_length
                                      , p_ud_data				:= p_ud_data
                                      , ud_type				:= VM_MEMORY_ACCESS
                                      );

	//look for an error
	if ( sd_retval <> VARANMANAGER_OK ) then
		State := _CreateDOFailed;
		VaranIn.SetState( State );
		return;
	end_if;
  end_if;

	//save pointer in array
	a_SpecialDO[ us_SpecialDOCnt ].p_Handle$^UDINT := ( p_ud_handle^ )$^UDINT;

  if b_PayloadSupport = FALSE then
	a_SpecialDO[ us_SpecialDOCnt ].p_Settings$^UDINT := ( p_ud_data^ )$^UDINT - VM_DO_OFFSET_WR;
  end_if;
	a_SpecialDO[ us_SpecialDOCnt ].p_DataWrite := ( p_ud_data^ )$^USINT;
	a_SpecialDO[ us_SpecialDOCnt ].us_Length := ud_length$USINT;

	us_SpecialDOCnt += 1;

END_FUNCTION //GLOBAL Varan_DataMover::AddVaranWrDO
(*
#if 0

//[#ENGLISH]
//[>ud_address]address for reading
//[>ud_length]max. 128 Byte access
//[>p_data]address  of pointer (pointer value is set)
FUNCTION GLOBAL Varan_DataMover::DirectAccessRead
VAR_INPUT
	ud_address		: UDINT;
	ud_length		: UDINT;
	p_data			: ^void;
END_VAR
VAR_OUTPUT
	sd_retval		: DINT;
END_VAR
VAR
	s_state			: t_DataMoverConfig;
	ud_timemark		: UDINT;
END_VAR

	if ( State = _ClassOk & s_DAData.b_Init = TRUE ) then

		//check length
		if ( ud_length > 128 | p_data = NIL ) then
			sd_retval := -101;
			return;
		end_if;

		LOCK_DA;

		//set command settings
		s_DAData.s_DAMove.ui_Length		:= ud_length$UINT;
		s_DAData.s_DAMove.ud_SourceAdd	:= ud_address;
		s_DAData.s_DAMove.ud_DestAdd	:= s_DAData.ud_DataAddressSub;		//max. 128 byte (1 varan data object)

		//write config data (because we need direct accesses in init)
		sd_retval := VARAN_iWriteMemoryDA	( uiManager		:= ud_VaranManagerNr
											, uiAddress		:= s_DAData.ud_CodeAddress
											, uiLen			:= sizeof( t_StructMove )
											, uiRetryTimeout:= s_DAData.ud_RetryTimeout
											, pvData		:= #s_DAData.s_DAMove
											, puiError		:= NIL
											);

		if ( sd_retval <> VARANMANAGER_OK ) then
			State := _DirectAccessFailed;
			VaranIn.SetState( State );
			UNLOCK_DA;
			return;
		end_if;

		//start list (write config data)
		s_Config.us_ControlReg.AdminEnable := TRUE;

		sd_retval := VARAN_iWriteMemoryDA	( uiManager		:= ud_VaranManagerNr
											, uiAddress		:= s_DAData.ud_StartAddress
											, uiLen			:= 1
											, uiRetryTimeout:= s_DAData.ud_RetryTimeout
											, pvData		:= #s_Config
											, puiError		:= NIL
											);

		if ( sd_retval <> VARANMANAGER_OK ) then
			State := _DirectAccessFailed;
			VaranIn.SetState( State );
			UNLOCK_DA;
			return;
		end_if;

		//poll if list is ready or timeout
		s_state.us_StateReg := 2#100;
		ud_timemark := Varanin.VaranIn.GetNsTime();
		while ( ( s_state.us_StateReg and 2#100 ) & ( VaranIn.VaranIn.GetNsTime() - ud_timemark ) < 50000 ) do

			sd_retval := VARAN_iReadMemoryDA	( uiManager		:= ud_VaranManagerNr
												, uiAddress		:= s_DAData.ud_StartAddress
												, uiLen			:= 4
												, uiRetryTimeout:= s_DAData.ud_RetryTimeout
												, pvData		:= #s_state
												, puiError		:= NIL
												);

			if ( sd_retval <> VARANMANAGER_OK ) then
				State := _DirectAccessFailed;
				VaranIn.SetState( State );
				UNLOCK_DA;
				return;
			end_if;
		end_while;

		//check timeout
		if ( s_state.us_StateReg and 2#100 ) then
			sd_retval := -102;
			Timeout += 1;
			UNLOCK_DA;
			return;
		end_if;

		if ( s_state.us_ErrorReg <> 0 ) then
			sd_retval := -102;
			State := _DirectAccessFailed;
			VaranIn.SetState( State );
			UNLOCK_DA;
			return;
		end_if;

		//read data
		sd_retval := VARAN_iReadMemoryDA	( uiManager		:= ud_VaranManagerNr
											, uiAddress		:= s_DAData.ud_DataAddress
											, uiLen			:= ud_length
											, uiRetryTimeout:= s_DAData.ud_RetryTimeout
											, pvData		:= p_data
											, puiError		:= NIL
											);

		if ( sd_retval <> VARANMANAGER_OK ) then
			State := _DirectAccessFailed;
			VaranIn.SetState( State );
			UNLOCK_DA;
			return;
		end_if;

		UNLOCK_DA;

	else
		sd_retval := -100;
	end_if;

END_FUNCTION //GLOBAL Varan_DataMover::DirectAccessRead

//[#ENGLISH]
//[>ud_address]address of write access
//[>ud_length]max. 128 Byte access
//[>p_data]address of pointer (pointer value is set)
FUNCTION GLOBAL Varan_DataMover::DirectAccessWrite
VAR_INPUT
	ud_address		: UDINT;
	ud_length		: UDINT;
	p_data			: ^void;
END_VAR
VAR_OUTPUT
	sd_retval		: DINT;
END_VAR
VAR
	s_state			: t_DataMoverConfig;
	ud_timemark		: UDINT;
END_VAR

	if ( State = _ClassOk & s_DAData.b_Init = TRUE ) then

		//check length
		if ( ud_length > 128 | p_data = NIL ) then
			sd_retval := -101;
			return;
		end_if;

		LOCK_DA;

		//set command settings
		s_DAData.s_DAMove.ui_Length		:= ud_length$UINT;
		s_DAData.s_DAMove.ud_SourceAdd	:= s_DAData.ud_DataAddressSub;		//max. 128 byte (1 varan data object)
		s_DAData.s_DAMove.ud_DestAdd	:= ud_address;

		//write config data (because we need direct accesses in init)
		sd_retval := VARAN_iWriteMemoryDA	( uiManager		:= ud_VaranManagerNr
											, uiAddress		:= s_DAData.ud_CodeAddress
											, uiLen			:= sizeof( t_StructMove )
											, uiRetryTimeout:= s_DAData.ud_RetryTimeout
											, pvData		:= #s_DAData.s_DAMove
											, puiError		:= NIL
											);

		if ( sd_retval <> VARANMANAGER_OK ) then
			State := _DirectAccessFailed;
			VaranIn.SetState( State );

			UNLOCK_DA;
			return;
		end_if;

		//write data
		sd_retval := VARAN_iWriteMemoryDA	( uiManager		:= ud_VaranManagerNr
											, uiAddress		:= s_DAData.ud_DataAddress
											, uiLen			:= ud_length
											, uiRetryTimeout:= s_DAData.ud_RetryTimeout
											, pvData		:= p_data
											, puiError		:= NIL
											);

		if ( sd_retval <> VARANMANAGER_OK ) then
			State := _DirectAccessFailed;
			VaranIn.SetState( State );
			UNLOCK_DA;
			return;
		end_if;

		//start list (write config data)
		s_Config.us_ControlReg.AdminEnable := TRUE;

		sd_retval := VARAN_iWriteMemoryDA	( uiManager		:= ud_VaranManagerNr
											, uiAddress		:= s_DAData.ud_StartAddress
											, uiLen			:= 1
											, uiRetryTimeout:= s_DAData.ud_RetryTimeout
											, pvData		:= #s_Config
											, puiError		:= NIL
											);

		if ( sd_retval <> VARANMANAGER_OK ) then
			State := _DirectAccessFailed;
			VaranIn.SetState( State );
			UNLOCK_DA;
			return;
		end_if;

		//poll if list is ready or timeout
		s_state.us_StateReg := 2#100;
		ud_timemark := Varanin.VaranIn.GetNsTime();
		while ( ( s_state.us_StateReg and 2#100 ) & ( VaranIn.VaranIn.GetNsTime() - ud_timemark ) < 1000000 ) do

			sd_retval := VARAN_iReadMemoryDA	( uiManager		:= ud_VaranManagerNr
												, uiAddress		:= s_DAData.ud_StartAddress
												, uiLen			:= 4
												, uiRetryTimeout:= s_DAData.ud_RetryTimeout
												, pvData		:= #s_state
												, puiError		:= NIL
												);

			if ( sd_retval <> VARANMANAGER_OK ) then
				State := _DirectAccessFailed;
				VaranIn.SetState( State );
				UNLOCK_DA;
				return;
			end_if;
		end_while;

		//check timeout
		if ( s_state.us_StateReg and 2#100 ) then
			sd_retval := -102;
			Timeout += 1;
			UNLOCK_DA;
			return;
		end_if;

		if ( s_state.us_ErrorReg <> 0 ) then
			sd_retval := -102;
			State := _DirectAccessFailed;
			VaranIn.SetState( State );
			UNLOCK_DA;
			return;
		end_if;

		UNLOCK_DA;

	else
		sd_retval := -100;
	end_if;

END_FUNCTION //GLOBAL Varan_DataMover::DirectAccessWrite

	//----------------------------------------------------------------------------------------------
	//Config mover
  s_Config.us_ControlReg                  := 0;
  s_Config.us_ControlReg.MoverEnable 			:= TRUE;
	s_Config.us_ControlReg.HoldOPError			:= TRUE;
	s_Config.us_ControlReg.HoldWBError			:= TRUE;
	s_Config.us_ControlReg.HoldTimeSliceError	:= TRUE;

	s_Config.ud_SyncTimeReg := VaranIn.GetVaranTime() / 2000;		//in µs

	//write config data (because we need direct accesses in init)
	sd_retval := VARAN_iWriteMemoryDA	( uiManager		:= ud_VaranManagerNr
										, uiAddress		:= ud_DeviceAddress+ CodeStartAddress
										, uiLen			:= sizeof( t_DataMoverConfig )
										, uiRetryTimeout:= VaranIn.GetRetryTimeout( ud_bytes := sizeof( t_DataMoverConfig ) )
										, pvData		:= #s_Config
										, puiError		:= NIL
										);

	if ( sd_retval <> VARANMANAGER_OK ) then
		State := _DirectAccessFailed;
		VaranIn.SetState( State );
		return;
	end_if;

	//----------------------------------------------------------------------------------------------
	//last 16 bytes are for direct access list
	s_ListSettings.ui_DAListStart 	:= TO_UINT( VM_DATAMOVER_HEADER + CodeSize - ( sizeof( t_StructMove ) + sizeof( t_StructEnd ) ) );
	s_ListSettings.ui_DAListEnd		:= TO_UINT( VM_DATAMOVER_HEADER + CodeSize - sizeof( t_StructEnd ) );
	s_ListSettings.ui_SyncListStart	:= 0;
	s_ListSettings.ui_SyncListEnd	:= 0;
	s_ListSettings.ui_AsyncListStart:= 0;
	s_ListSettings.ui_AsyncListEnd	:= 0;

	//write list config data (because we need direct accesses in init)
	sd_retval := VARAN_iWriteMemoryDA	( uiManager		:= ud_VaranManagerNr
										, uiAddress		:= ud_DeviceAddress + CodeStartAddress + VM_LIST_CONFIG_OFFSET
										, uiLen			:= sizeof( t_ListConfig )
										, uiRetryTimeout:= VaranIn.GetRetryTimeout( ud_bytes := sizeof( t_ListConfig ) )
										, pvData		:= #s_ListSettings
										, puiError		:= NIL
										);

	if ( sd_retval <> VARANMANAGER_OK ) then
		State := _DirectAccessFailed;
		VaranIn.SetState( State );
		return;
	end_if;

	//----------------------------------------------------------------------------------------------
	//settings for direct accesses
	s_DAData.ud_CodeAddress			:= ud_DeviceAddress + CodeStartAddress + s_ListSettings.ui_DAListStart;
	s_DAData.ud_DataAddress			:= ud_DeviceAddress + DPRAM_StartAddress + DPRAM_Size - 128;
	s_DAData.ud_RetryTimeout		:= VaranIn.GetRetryTimeout( ud_bytes := 128 );
	s_DAData.ud_DataAddressSub		:= DPRAM_StartAddress_SUBBus + DPRAM_Size - 128;
	s_DAData.ud_StartAddress		:= ud_DeviceAddress + CodeStartAddress + t_DataMoverConfig.us_ControlReg;
	s_DAData.s_DAMove.us_Command	:= VM_DATAMOVER_MOVE_OP;

	//write end command to da list
	ui_EndAddressOff := TO_UINT( s_ListSettings.ui_DAListStart + sizeof( t_StructMove ) );

	sd_retval := VARAN_iWriteMemoryDA	( uiManager		:= ud_VaranManagerNr
										, uiAddress		:= s_DAData.ud_CodeAddress + sizeof( t_StructMove )
										, uiLen			:= sizeof( t_StructEnd )
										, uiRetryTimeout:= VaranIn.GetRetryTimeout( ud_bytes := sizeof( t_StructEnd ) )
										, pvData		:= #s_End
										, puiError		:= NIL
										);

	//look for error
	if ( sd_retval <> VARANMANAGER_OK ) then
		State := _DirectAccessFailed;
		VaranIn.SetState( State );
		return;
	end_if;

	s_DAData.b_Init := TRUE;

#endif

*)

FUNCTION GLOBAL Varan_DataMover::SafetyMoverDisable

  // tell the OS that we configured the Mover
  if ( ( pHardwareTree <> NIL ) & ( pHardwareTree^.udVersion >= 16#1002 ) ) then
    //LanSte 20.11.2013 17:19 This call will cause in Access Exception if the info block of the Module is incorrectly configured
    //LanSte 20.11.2013 17:20 Check if FPGA Info Block exists and contains an entry for DevType = 0E60
    HWT_iDataMoverDisable(ud_VaranManagerNr, VaranIn.GetPointer2ObjectPath());
  end_if;

END_FUNCTION

FUNCTION GLOBAL Varan_DataMover::SafetyMoverEnable
	VAR_INPUT
		MoverActive 	: DINT;
	END_VAR

  if ( ( pHardwareTree <> NIL ) & ( pHardwareTree^.udVersion >= 16#1002 ) ) then
    //LanSte 20.11.2013 17:19 This call will cause in Access Exception if the info block of the Module is incorrectly configured
    //LanSte 20.11.2013 17:20 Check if FPGA Info Block exists and contains an entry for DevType = 0E60
    HWT_iDataMoverEnable(ud_VaranManagerNr, VaranIn.GetPointer2ObjectPath(), (#s_Config.us_ControlReg)$^USINT, (#us_ControlRd)$^USINT, MoverActive$UDINT, #ud_AdminCnt);
  end_if;

END_FUNCTION

FUNCTION GLOBAL Varan_DataMover::SafetyMoverConfigured

  // check how many DPRAM is reserved by HW-Classes => OS uses the rest (if it's enough)

  // we start with the last entry in the DPRAM and work backwards (if there is no entry for it)
  if s_Set_ASY_WR.us_DOCount then
    // we have asynchronous write DOs => <reserved memory> = <offset of asy wr DOs inside DPRAM> + <number of DOs - 1> * <size of each DO> + <size of last DO>
    ud_MoverDPRAM_Used := (s_Set_ASY_WR.ui_DPRAMOffset - DPRAM_StartAddress) + (s_Set_ASY_WR.us_DOCount-1) * 128 + a_DO_ASY_WR[s_Set_ASY_WR.us_DOCount-1].us_Length;
  elsif s_Set_ASY_RD.us_DOCount then
    // we have asynchronous read DOs => <reserved memory> = <offset of asy rd DOs inside DPRAM> + <number of DOs - 1> * <size of each DO> + <size of last DO>
    ud_MoverDPRAM_Used := (s_Set_ASY_RD.ui_DPRAMOffset - DPRAM_StartAddress) + (s_Set_ASY_RD.us_DOCount-1) * 128 + a_DO_ASY_RD[s_Set_ASY_RD.us_DOCount-1].us_Length;
  elsif s_Set_ISO_WR.us_DOCount then
    // we have asynchronous write DOs => <reserved memory> = <offset of asy wr DOs inside DPRAM> + <number of DOs - 1> * <size of each DO> + <size of last DO>
    ud_MoverDPRAM_Used := (s_Set_ISO_WR.ui_DPRAMOffset - DPRAM_StartAddress) + (s_Set_ISO_WR.us_DOCount-1) * 128 + a_DO_ISO_WR[s_Set_ISO_WR.us_DOCount-1].us_Length;
  elsif s_Set_ISO_RD.us_DOCount then
    // we have asynchronous write DOs => <reserved memory> = <offset of asy wr DOs inside DPRAM> + <number of DOs - 1> * <size of each DO> + <size of last DO>
    ud_MoverDPRAM_Used := (s_Set_ISO_RD.ui_DPRAMOffset - DPRAM_StartAddress) + (s_Set_ISO_RD.us_DOCount-1) * 128 + a_DO_ISO_RD[s_Set_ISO_RD.us_DOCount-1].us_Length;
  else
    ud_MoverDPRAM_Used := 0;
  end_if;

  // tell the OS that we configure the DAs in a second
  if ( ( pHardwareTree <> NIL ) & ( pHardwareTree^.udVersion >= 16#1002 ) ) then
    HWT_iDataMoverConfigured(ud_VaranManagerNr, VaranIn.GetPointer2ObjectPath(), ud_MoverDPRAM_Used);
  end_if;

END_FUNCTION

//#WP003 start
FUNCTION GLOBAL Varan_DataMover::CreateDOs
  VAR
    i           : USINT;
    sd_retval		: DINT;
  END_VAR

  //set back length of code (2nd callback get this infos again)
  ui_ASYByteCount := 0;
  ui_ISOByteCount := 0;
  s_DAData.b_Init := FALSE;

  //look if we have to create ISO Rd DO(s)
  if ( s_Set_ISO_RD.us_DOCount ) then
		for i := 0 to (s_Set_ISO_RD.us_DOCount - 1) do
      if b_PayloadSupport then
        sd_retval := VaranIn.AddRdPayloadDO(ud_dol_type   := VARAN_DOL_ISO
                                    , p_ud_handle   := ( #a_DO_ISO_RD[i].p_Handle)$^UDINT
                                    , ud_offset_read      := s_Set_ISO_RD.ui_DPRAMOffset + ( i * 128 )
                                    , ud_length_read      := a_DO_ISO_RD[i].us_Length
                                    , p_ud_data_read      := ( #a_DO_ISO_RD[i].p_DataRead)$^UDINT
                                    , ud_type             := VM_MEMORY_ACCESS
                                    , ud_priority         := a_DO_ISO_RD[i].ud_Priority
                                    , ud_WritePayloadType := 1);

        //look for an error
        if ( sd_retval <> VARANMANAGER_OK ) then
          State := _CreateDOFailed;
          VaranIn.SetState( State );
          return;
        end_if;
      else
      //create DO
        sd_retval := VaranIn.VaranIn.AddRdDO( p_us_position_info  := p_NodeString
                                            , ud_dol_type         := VARAN_DOL_ISO
                                            , p_ud_handle         := ( #a_DO_ISO_RD[i].p_Handle )$^UDINT
                                            , ud_address          := s_Set_ISO_RD.ui_DPRAMOffset + ( i * 128 )
                                            , ud_length           := a_DO_ISO_RD[i].us_Length
                                            , p_ud_data           := ( #a_DO_ISO_RD[i].p_DataRead )$^UDINT
                                            , ud_type             := VM_MEMORY_ACCESS OR a_DO_ISO_RD[i].ud_Priority
                                          );

      //look for an error
      if ( sd_retval <> VARANMANAGER_OK ) then
        State := _CreateDOFailed;
        VaranIn.SetState( State );
        return;
      end_if;

      //set settings pointer
      a_DO_ISO_RD[i].p_Settings$^USINT := a_DO_ISO_RD[i].p_DataRead - VM_DO_OFFSET_RD;
      end_if;

      //reset length of DO
      a_DO_ISO_RD[i].us_Length := 0;

      // Save Handle to external variable
      if a_DO_ISO_RD[i].p_UserDOHandle then
        a_DO_ISO_RD[i].p_UserDOHandle^ := a_DO_ISO_RD[i].p_Handle$UDINT;
      end_if;

    end_for;
  end_if;

  //look if we have to create ISO Wr DO(s)
  if ( s_Set_ISO_Wr.us_DOCount ) then
		for i := 0 to (s_Set_ISO_Wr.us_DOCount - 1) do

      //create DO
      if b_PayloadSupport then
        sd_retval := VaranIn.AddWrPayloadDO(ud_dol_type   := VARAN_DOL_ISO
                                    , p_ud_handle   := ( #a_DO_ISO_WR[i].p_Handle)$^UDINT
                                    , ud_offset_write     := s_Set_ISO_WR.ui_DPRAMOffset + ( i * 128 )
                                    , ud_length_write     := a_DO_ISO_WR[i].us_Length
                                    , p_ud_data_write     := ( #a_DO_ISO_WR[i].p_DataWrite)$^UDINT
                                    , ud_type             := VM_MEMORY_ACCESS
                                    , ud_priority         := a_DO_ISO_WR[i].ud_Priority
                                    , ud_WritePayloadType := 1);

        //look for an error
        if ( sd_retval <> VARANMANAGER_OK ) then
          State := _CreateDOFailed;
          VaranIn.SetState( State );
          return;
        end_if;
      else
        sd_retval := VaranIn.VaranIn.AddWrDO( p_us_position_info  := p_NodeString
                                            , ud_dol_type         := VARAN_DOL_ISO
                                            , p_ud_handle         := ( #a_DO_ISO_WR[i].p_Handle )$^UDINT
                                            , ud_address          := s_Set_ISO_WR.ui_DPRAMOffset + ( i * 128 )
                                            , ud_length           := a_DO_ISO_WR[i].us_Length
                                            , p_ud_data           := ( #a_DO_ISO_WR[i].p_DataWrite )$^UDINT
                                            , ud_type             := VM_MEMORY_ACCESS OR a_DO_ISO_WR[i].ud_Priority
                                          );

      //look for an error
      if ( sd_retval <> VARANMANAGER_OK ) then
        State := _CreateDOFailed;
        VaranIn.SetState( State );
        return;
      end_if;

      //set settings pointer
      a_DO_ISO_WR[i].p_Settings$^USINT := a_DO_ISO_WR[i].p_DataWrite - VM_DO_OFFSET_WR;
      end_if;

      //reset length of DO
      a_DO_ISO_WR[i].us_Length := 0;

      // Save Handle to external variable
      if a_DO_ISO_WR[i].p_UserDOHandle then
        a_DO_ISO_WR[i].p_UserDOHandle^ := a_DO_ISO_WR[i].p_Handle$UDINT;
      end_if;

    end_for;
  end_if;

  //look if we have to create ASY Rd DO(s)
  if ( s_Set_ASY_RD.us_DOCount ) then
		for i := 0 to (s_Set_ASY_RD.us_DOCount - 1) do

      //create DO
      if b_PayloadSupport then
        sd_retval := VaranIn.AddRdPayloadDO(ud_dol_type   := VARAN_DOL_ASY
                                    , p_ud_handle   := ( #a_DO_ASY_RD[i].p_Handle)$^UDINT
                                    , ud_offset_read      := s_Set_ASY_RD.ui_DPRAMOffset + ( i * 128 )
                                    , ud_length_read      := a_DO_ASY_RD[i].us_Length
                                    , p_ud_data_read      := ( #a_DO_ASY_RD[i].p_DataRead)$^UDINT
                                    , ud_type             := VM_MEMORY_ACCESS
                                    , ud_priority         := a_DO_ASY_RD[i].ud_Priority
                                    , ud_WritePayloadType := 1);

        //look for an error
        if ( sd_retval <> VARANMANAGER_OK ) then
          State := _CreateDOFailed;
          VaranIn.SetState( State );
          return;
        end_if;
      else
        sd_retval := VaranIn.VaranIn.AddRdDO( p_us_position_info  := p_NodeString
                                            , ud_dol_type         := VARAN_DOL_ASY
                                            , p_ud_handle         := ( #a_DO_ASY_RD[i].p_Handle )$^UDINT
                                            , ud_address          := s_Set_ASY_RD.ui_DPRAMOffset + ( i * 128 )
                                            , ud_length           := a_DO_ASY_RD[i].us_Length
                                            , p_ud_data           := ( #a_DO_ASY_RD[i].p_DataRead )$^UDINT
                                            , ud_type             := VM_MEMORY_ACCESS OR a_DO_ASY_RD[i].ud_Priority
                                          );

      //look for an error
      if ( sd_retval <> VARANMANAGER_OK ) then
        State := _CreateDOFailed;
        VaranIn.SetState( State );
        return;
      end_if;

      //set settings pointer
      a_DO_ASY_RD[i].p_Settings$^USINT := a_DO_ASY_RD[i].p_DataRead - VM_DO_OFFSET_RD;
      end_if;

      //reset length of DO
      a_DO_ASY_RD[i].us_Length := 0;

      // Save Handle to external variable
      if a_DO_ASY_RD[i].p_UserDOHandle then
        a_DO_ASY_RD[i].p_UserDOHandle^ := a_DO_ASY_RD[i].p_Handle$UDINT;
      end_if;

    end_for;
  end_if;

  //look if we have to create ASY Wr DO(s)
  if ( s_Set_ASY_WR.us_DOCount ) then
		for i := 0 to (s_Set_ASY_WR.us_DOCount - 1) do

      //create DO

      if b_PayloadSupport then
        sd_retval := VaranIn.AddWrPayloadDO(ud_dol_type   := VARAN_DOL_ASY
                                    , p_ud_handle   := ( #a_DO_ASY_WR[i].p_Handle)$^UDINT
                                    , ud_offset_write     := s_Set_ASY_WR.ui_DPRAMOffset + ( i * 128 )
                                    , ud_length_write     := a_DO_ASY_WR[i].us_Length
                                    , p_ud_data_write     := ( #a_DO_ASY_WR[i].p_DataWrite)$^UDINT
                                    , ud_type             := VM_MEMORY_ACCESS
                                    , ud_priority         := a_DO_ASY_WR[i].ud_Priority
                                    , ud_WritePayloadType := 1);

        //look for an error
        if ( sd_retval <> VARANMANAGER_OK ) then
          State := _CreateDOFailed;
          VaranIn.SetState( State );
          return;
        end_if;
      else
        sd_retval := VaranIn.VaranIn.AddWrDO( p_us_position_info  := p_NodeString
                                            , ud_dol_type         := VARAN_DOL_ASY
                                            , p_ud_handle         := ( #a_DO_ASY_WR[i].p_Handle )$^UDINT
                                            , ud_address          := s_Set_ASY_WR.ui_DPRAMOffset + ( i * 128 )
                                            , ud_length           := a_DO_ASY_WR[i].us_Length
                                            , p_ud_data           := ( #a_DO_ASY_WR[i].p_DataWrite )$^UDINT
                                            , ud_type             := VM_MEMORY_ACCESS OR a_DO_ASY_WR[i].ud_Priority
                                          );

      //look for an error
      if ( sd_retval <> VARANMANAGER_OK ) then
        State := _CreateDOFailed;
        VaranIn.SetState( State );
        return;
      end_if;

      //set settings pointer
      a_DO_ASY_WR[i].p_Settings$^USINT := a_DO_ASY_WR[i].p_DataWrite - VM_DO_OFFSET_WR;
      end_if;

      //reset length of DO
      a_DO_ASY_WR[i].us_Length := 0;

      // Save Handle to external variable
      if a_DO_ASY_WR[i].p_UserDOHandle then
        a_DO_ASY_WR[i].p_UserDOHandle^ := a_DO_ASY_WR[i].p_Handle$UDINT;
      end_if;

    end_for;
  end_if;

  //mark as created well
  DO_Created := true;

END_FUNCTION
//#WP003 end

FUNCTION GLOBAL Varan_DataMover::AddMoveISO
VAR_INPUT
  SourceAddr 	: HDINT;
  DestAddr 	: HDINT;
  MoveLen 	: UDINT;
  pEnable 	: ^USINT;
  udPriority 	: UDINT;
END_VAR
VAR_OUTPUT
  sd_retval 	: DINT;
END_VAR
VAR
	p_Mov			    : ^t_StructMove;
	p_MovEn			  : ^t_StructMoveEn;
	ud_en_add		  : UDINT;
END_VAR

  if pEnable then
    //for enable byte
    sd_retval := GetMemoryISOWr	( p_add		:= #ud_en_add
                  , p_data	:= pEnable
                  , ud_len	:= 1
                  , ud_Priority := udPriority
                  );

    if ( sd_retval <> VARANMANAGER_OK ) then
      return;
    end_if;

    //give back address of enable byte
    ( ( ( pEnable$^UDINT )^ )$^USINT )^ := 0;

  end_if;

	//save opcodes in class
	if ( p_ISOMoverCode = NIL ) then
		//allocate memory
		p_ISOMoverCode$^void := To_StdLib.Malloc( s_Set_ISO_RD.ui_DPRAMSize + s_Set_ISO_WR.ui_DPRAMSize );

		if ( p_ISOMoverCode  = NIL ) then
			State := _MemoryFault;
			sd_retval := -103;
			VaranIn.SetState( State );
			return;
		end_if;
	end_if;

	//first check length
	if ( CheckLengthOfCode() = FALSE ) then
		sd_retval := -102;
		return;
	end_if;

  if pEnable then
    //check size of free memory
    if (( ui_ISOByteCount + sizeof( t_StructMoveEn )) > ( s_Set_ISO_RD.ui_DPRAMSize + s_Set_ISO_WR.ui_DPRAMSize )) then
      State := _MemoryFault;
      sd_retval := -102;
      VaranIn.SetState( State );
      return;
    end_if;

    //get right pointer
    p_MovEn := p_ISOMoverCode + ui_ISOByteCount;

    p_MovEn^.us_Command 		:= VM_DATAMOVER_MOVE_EN_OP;
    p_MovEn^.ui_Length		:= MoveLen$UINT;
    p_MovEn^.us_Length		:= ( MoveLen shr 16 )$USINT;
    p_MovEn^.ud_SourceAdd		:= SourceAddr;
    p_MovEn^.ud_DestAdd		:= DestAddr;
    p_MovEn^.ud_EnableAddByte	:= ud_en_add;

    ui_ISOByteCount += sizeof( t_StructMoveEn );
  else
    //check size of free memory
    if (( ui_ISOByteCount + sizeof( t_StructMove )) > ( s_Set_ISO_RD.ui_DPRAMSize + s_Set_ISO_WR.ui_DPRAMSize )) then
      State := _MemoryFault;
      sd_retval := -102;
      VaranIn.SetState( State );
      return;
    end_if;

    //get right pointer
    p_Mov := p_ISOMoverCode + ui_ISOByteCount;

    p_Mov^.us_Command 		:= VM_DATAMOVER_MOVE_OP;
    p_Mov^.ui_Length		:= MoveLen$UINT;
    p_Mov^.us_Length		:= ( MoveLen shr 16 )$USINT;
    p_Mov^.ud_SourceAdd		:= SourceAddr;
    p_Mov^.ud_DestAdd		:= DestAddr;

    ui_ISOByteCount += sizeof( t_StructMove );
  end_if;

	sd_retval := VARANMANAGER_OK;

END_FUNCTION

FUNCTION GLOBAL Varan_DataMover::AddMoveASY
	VAR_INPUT
		SourceAddr 	: HDINT;
		DestAddr 	: HDINT;
		MoveLen 	: UDINT;
		pEnable 	: ^USINT;
		udPriority 	: UDINT;
	END_VAR
	VAR_OUTPUT
		sd_retval 	: DINT;
	END_VAR
VAR
	p_Mov			    : ^t_StructMove;
	p_MovEn			  : ^t_StructMoveEn;
	ud_en_add		  : UDINT;
END_VAR

  if pEnable then
    //for enable byte
    sd_retval := GetMemoryASYWr	( p_add		:= #ud_en_add
                  , p_data	:= pEnable
                  , ud_len	:= 1
                  , ud_Priority := udPriority
                  );

    if ( sd_retval <> VARANMANAGER_OK ) then
      return;
    end_if;

    //give back address of enable byte
    ( ( ( pEnable$^UDINT )^ )$^USINT )^ := 0;

  end_if;

	//save opcodes in class
	if ( p_ASYMoverCode = NIL ) then
		//allocate memory
		p_ASYMoverCode$^void := To_StdLib.Malloc( s_Set_ASY_RD.ui_DPRAMSize + s_Set_ASY_WR.ui_DPRAMSize );

		if ( p_ASYMoverCode  = NIL ) then
			State := _MemoryFault;
			sd_retval := -103;
			VaranIn.SetState( State );
			return;
		end_if;
	end_if;

	//first check length
	if ( CheckLengthOfCode() = FALSE ) then
		sd_retval := -102;
		return;
	end_if;

  if pEnable then
    //check size of free memory
    if (( ui_ASYByteCount + sizeof( t_StructMoveEn )) > ( s_Set_ASY_RD.ui_DPRAMSize + s_Set_ASY_WR.ui_DPRAMSize )) then
      State := _MemoryFault;
      sd_retval := -102;
      VaranIn.SetState( State );
      return;
    end_if;

    //get right pointer
    p_MovEn := p_ASYMoverCode + ui_ASYByteCount;

    p_MovEn^.us_Command 		:= VM_DATAMOVER_MOVE_EN_OP;
    p_MovEn^.ui_Length		:= MoveLen$UINT;
    p_MovEn^.us_Length		:= ( MoveLen shr 16 )$USINT;
    p_MovEn^.ud_SourceAdd		:= SourceAddr;
    p_MovEn^.ud_DestAdd		:= DestAddr;
    p_MovEn^.ud_EnableAddByte	:= ud_en_add;

    ui_ASYByteCount += sizeof( t_StructMoveEn );
  else
    //check size of free memory
    if (( ui_ASYByteCount + sizeof( t_StructMove )) > ( s_Set_ASY_RD.ui_DPRAMSize + s_Set_ASY_WR.ui_DPRAMSize )) then
      State := _MemoryFault;
      sd_retval := -102;
      VaranIn.SetState( State );
      return;
    end_if;

    //get right pointer
    p_Mov := p_ASYMoverCode + ui_ASYByteCount;

    p_Mov^.us_Command 		:= VM_DATAMOVER_MOVE_OP;
    p_Mov^.ui_Length		:= MoveLen$UINT;
    p_Mov^.us_Length		:= ( MoveLen shr 16 )$USINT;
    p_Mov^.ud_SourceAdd		:= SourceAddr;
    p_Mov^.ud_DestAdd		:= DestAddr;

    ui_ASYByteCount += sizeof( t_StructMove );
  end_if;

	sd_retval := VARANMANAGER_OK;

END_FUNCTION
